// SIMATIC S7-200 project (STEP 7-Micro/WIN), CPU 224XP REL 02.01

SYMBOL_TABLE USER1
star             I0.0
s_top            I0.1
den_xanh1        Q0.1
den_vàng1        Q0.2
den_do1          Q0.3
den_xanh2        Q0.5
den_vang2        Q0.6
den_do2          Q0.7
bien             M0.0
END_SYMBOL_TABLE

ORGANIZATION_BLOCK MAIN:OB1
TITLE=PROGRAM COMMENTS
BEGIN
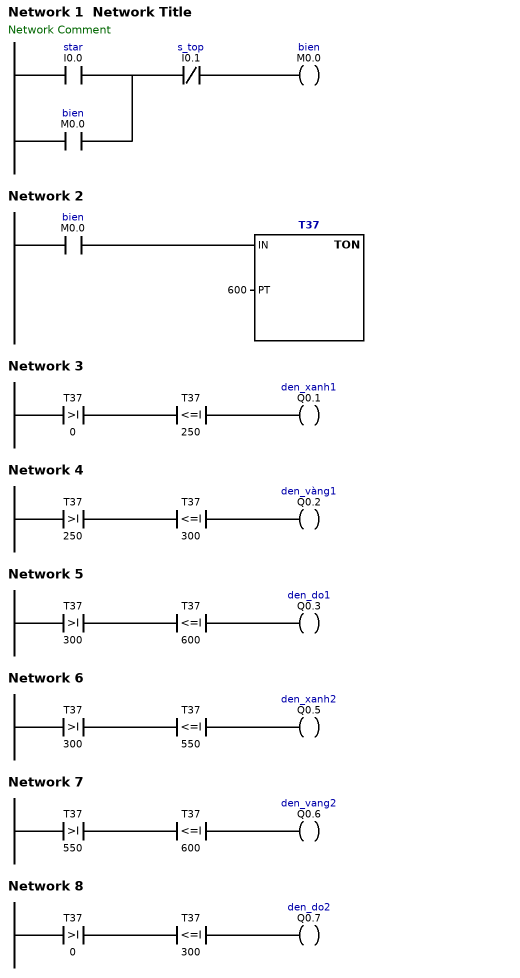
Network 1 // Network Title
// Network Comment
LD     star:I0.0
O      bien:M0.0
AN     s_top:I0.1
=      bien:M0.0
Network 2
LD     bien:M0.0
TON    T37, 600
Network 3
LDW>   T37, 0
AW<=   T37, 250
=      den_xanh1:Q0.1
Network 4
LDW>   T37, 250
AW<=   T37, 300
=      den_vàng1:Q0.2
Network 5
LDW>   T37, 300
AW<=   T37, 600
=      den_do1:Q0.3
Network 6
LDW>   T37, 300
AW<=   T37, 550
=      den_xanh2:Q0.5
Network 7
LDW>   T37, 550
AW<=   T37, 600
=      den_vang2:Q0.6
Network 8
LDW>   T37, 0
AW<=   T37, 300
=      den_do2:Q0.7
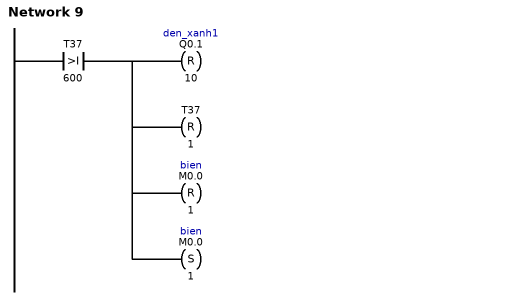
Network 9
LDW>   T37, 600
R      den_xanh1:Q0.1, 10
R      T37, 1
R      bien:M0.0, 1
S      bien:M0.0, 1
END_ORGANIZATION_BLOCK
